{attribute 'qualified_only'}
{attribute 'strict'}
{attribute 'to_string'}
TYPE CSVWriteMode :
(
	keyence := 0,
	massa	:= 1,
	sonar	:= 2,
	script	:= 3
);
END_TYPE

(* stored: Version 1.1.0.1, ProductVersion 3.1.4026.12
   DUT CSVWriteMode: Id {edefb3b5-a8a0-45a9-a11f-0c98204575f6} *)
